// TIA Portal project "babu_SinglePBOnOff" (V15)

(* hardware
DEVICE "S7-1200 station_1"  S7-1200 Station
   slot 0: "Rack_0"  S7-1200 Rack  Rack  V1.0
   slot 1: "PLC_1"  CPU 1214C DC/DC/DC  6ES7 214-1AG40-0XB0  V4.2
*)

// ===== PLC "PLC_1"  CPU 1214C DC/DC/DC =====

VAR_GLOBAL   // PLC tag table "Default tag table"
   "PUSH BUTTON" AT %M0.0 : Bool;
   "TEMP" AT %M0.1 : Bool;
   "OUTPUT" AT %Q0.0 : Bool;
   "OUTPUT MEM" AT %M0.2 : Bool;
   "PREVIOUS MEM" AT %M0.3 : Bool;
   "TEMP 1" AT %M0.4 : Bool;
   "OUTPUT 1" AT %Q0.1 : Bool;
   "NC" AT %M0.5 : Bool;
END_VAR

ORGANIZATION_BLOCK "Main"   // OB1, LAD, ProgramCycle
TITLE = "Main Program Sweep (Cycle)"
{ S7_Optimized_Access := 'TRUE' }
VERSION : 0.1
   VAR_INPUT
      Initial_Call : Bool;   // Initial call of this OB
      Remanence : Bool;   // =True, if remanent data are available
   END_VAR
   VAR_TEMP   // added for the SCL form of the ladder/FBD networks
      _w1 : Bool;
   END_VAR
BEGIN

REGION Network 1
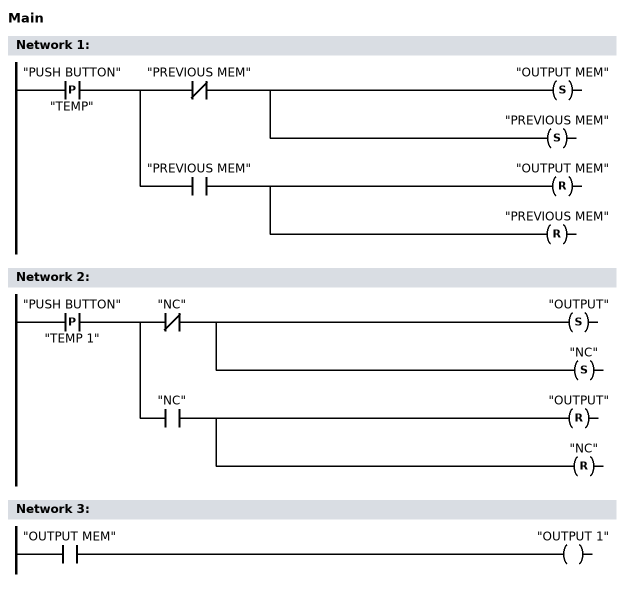
   RUNG wire#powerrail
      P_Contact(operand := "PUSH BUTTON", bit := "TEMP")
      wire#w1
      I_Contact( "PREVIOUS MEM" )
      wire#w2
      S_Coil( "OUTPUT MEM" )
   END_RUNG
   RUNG wire#w2
      S_Coil( "PREVIOUS MEM" )
   END_RUNG
   RUNG wire#w1
      Contact( "PREVIOUS MEM" )
      wire#w3
      R_Coil( "OUTPUT MEM" )
   END_RUNG
   RUNG wire#w3
      R_Coil( "PREVIOUS MEM" )
   END_RUNG
   // the same network as SCL:
   #_w1 := "PUSH BUTTON" AND NOT "TEMP";   // rising edge of "PUSH BUTTON"
   "TEMP" := "PUSH BUTTON";
   IF #_w1 AND NOT "PREVIOUS MEM" THEN
       "OUTPUT MEM" := TRUE;
       "PREVIOUS MEM" := TRUE;
   END_IF;
   IF #_w1 AND "PREVIOUS MEM" THEN
       "OUTPUT MEM" := FALSE;
       "PREVIOUS MEM" := FALSE;
   END_IF;
END_REGION

REGION Network 2
   RUNG wire#powerrail
      P_Contact(operand := "PUSH BUTTON", bit := "TEMP 1")
      wire#w1
      I_Contact( "NC" )
      wire#w2
      S_Coil( "OUTPUT" )
   END_RUNG
   RUNG wire#w2
      S_Coil( "NC" )
   END_RUNG
   RUNG wire#w1
      Contact( "NC" )
      wire#w3
      R_Coil( "OUTPUT" )
   END_RUNG
   RUNG wire#w3
      R_Coil( "NC" )
   END_RUNG
   // the same network as SCL:
   #_w1 := "PUSH BUTTON" AND NOT "TEMP 1";   // rising edge of "PUSH BUTTON"
   "TEMP 1" := "PUSH BUTTON";
   IF #_w1 AND NOT "NC" THEN
       "OUTPUT" := TRUE;
       "NC" := TRUE;
   END_IF;
   IF #_w1 AND "NC" THEN
       "OUTPUT" := FALSE;
       "NC" := FALSE;
   END_IF;
END_REGION

REGION Network 3
   RUNG wire#powerrail
      Contact( "OUTPUT MEM" )
      Coil( "OUTPUT 1" )
   END_RUNG
   // the same network as SCL:
   "OUTPUT 1" := "OUTPUT MEM";
END_REGION
END_ORGANIZATION_BLOCK